{attribute 'qualified_only'}
VAR_GLOBAL
	Device_type															: ST_CAN_Object := (Name:='Device type', 														Index:=16#1000, 			 			Writeable:=FALSE);
	Error_register														: ST_CAN_Object := (Name:='Error register', 													Index:=16#1001, 			 Length:=1, Writeable:=FALSE);
	Manufacturer_status_register										: ST_CAN_Object := (Name:='Manufacturer status register', 										Index:=16#1002, 			 			Writeable:=FALSE);
	Pre_defined_error_field_Number_of_errors							: ST_CAN_Object := (Name:='Pre-defined error field_Number of errors',							Index:=16#1003, 			 Length:=1, 										SubElements:=E_SubElement_types.With_list);
	Pre_defined_error_field_Standard_error_field_1						: ST_CAN_Object := (Name:='Pre-defined error field_Standard error field 1',						Index:=16#1003, Subindex:=1, 			Writeable:=FALSE,						SubElements:=E_SubElement_types.List_element);
	COB_ID_SYNC															: ST_CAN_Object := (Name:='COB-ID SYNC',														Index:=16#1005, 			 			Writeable:=FALSE, Default_Value:=16#80);
	Communication_cycle_period											: ST_CAN_Object := (Name:='Communication cycle period',											Index:=16#1006);
	Synchronous_window_length											: ST_CAN_Object := (Name:='Synchronous window length',											Index:=16#1007);
	Manufacturer_device_name											: ST_CAN_Object := (Name:='Manufacturer device name', 											Index:=16#1008, 			 Length:=0, Writeable:=FALSE);
	Manufacturer_hardware_version										: ST_CAN_Object := (Name:='Manufacturer hardware version',										Index:=16#1009, 			 Length:=0, Writeable:=FALSE);
	Manufacturer_software_version										: ST_CAN_Object := (Name:='Manufacturer software version',										Index:=16#100A, 			 Length:=0, Writeable:=FALSE);
	Guard_time															: ST_CAN_Object := (Name:='Guard time', 														Index:=16#100C, 			 Length:=2, Writeable:=FALSE);
	Life_time_factor													: ST_CAN_Object := (Name:='Life time factor', 													Index:=16#100D, 			 Length:=1, Writeable:=FALSE);
	store_parameters_highest_sub_index_supported						: ST_CAN_Object := (Name:='store parameters_highest sub-index supported', 						Index:=16#1010, 			 Length:=1, Writeable:=FALSE, Default_Value:=4, 	SubElements:=E_SubElement_types.With_fix_subelements);
	store_parameters_save_all_parameters								: ST_CAN_Object := (Name:='store parameters_save all parameters', 								Index:=16#1010, Subindex:=1, 													SubElements:=E_SubElement_types.Fix_subelement);
	store_parameters_save_communication_parameters						: ST_CAN_Object := (Name:='store parameters_save communication parameters', 					Index:=16#1010, Subindex:=2, 													SubElements:=E_SubElement_types.Fix_subelement);
	store_parameters_save_application_parameters						: ST_CAN_Object := (Name:='store parameters_save application parameters', 						Index:=16#1010, Subindex:=3, 													SubElements:=E_SubElement_types.Fix_subelement);
	store_parameters_save_manufacture_label								: ST_CAN_Object := (Name:='store parameters_save manufacture label', 							Index:=16#1010, Subindex:=4, 													SubElements:=E_SubElement_types.Fix_subelement);
	restore_default_parameters_highest_sub_index_supported				: ST_CAN_Object := (Name:='restore default parameters_highest sub-index supported', 			Index:=16#1011, 			 Length:=1, Writeable:=FALSE, Default_Value:=4, 	SubElements:=E_SubElement_types.With_fix_subelements);
	restore_default_parameters_restore_all_default_parameters			: ST_CAN_Object := (Name:='restore default parameters_restore all default parameters', 			Index:=16#1011, Subindex:=1,													SubElements:=E_SubElement_types.Fix_subelement);
	restore_default_parameters_restore_communication_default_parameters	: ST_CAN_Object := (Name:='restore default parameters_restore communication default parameters',Index:=16#1011, Subindex:=2,													SubElements:=E_SubElement_types.Fix_subelement);
	restore_default_parameters_restore_application_default_parameters	: ST_CAN_Object := (Name:='restore default parameters_restore application default parameters', 	Index:=16#1011, Subindex:=3,													SubElements:=E_SubElement_types.Fix_subelement);
	restore_default_parameters_restore_default_manufacture_label		: ST_CAN_Object := (Name:='restore default parameters_restore default manufacture label', 		Index:=16#1011, Subindex:=4,													SubElements:=E_SubElement_types.Fix_subelement);
	COB_ID_time_stamp_message											: ST_CAN_Object := (Name:='COB-ID time stamp message', 											Index:=16#1012);
	High_resolution_time_stamp											: ST_CAN_Object := (Name:='High resolution time stamp', 										Index:=16#1013);
	COB_ID_emergency_message											: ST_CAN_Object := (Name:='COB-ID emergency message', 											Index:=16#1014);
	Inhibit_time_emergency_message										: ST_CAN_Object := (Name:='Inhibit time emergency message', 									Index:=16#1015, 			 Length:=2);
	Consumer_heartbeat_time_highest_sub_index_supported					: ST_CAN_Object := (Name:='Consumer heartbeat time_highest sub-index supported', 				Index:=16#1016, 			 Length:=1, 										SubElements:=E_SubElement_types.With_list);
	Consumer_heartbeat_time_1											: ST_CAN_Object := (Name:='Consumer heartbeat time 1',											Index:=16#1016, Subindex:=1, 													SubElements:=E_SubElement_types.List_element);
	Producer_heartbeat_time												: ST_CAN_Object := (Name:='Producer heartbeat time', 											Index:=16#1017, 			 Length:=2);
	Identity_object_Highest_sub_index_supported							: ST_CAN_Object := (Name:='Identity object_Highest sub-index supported', 						Index:=16#1018, 			 Length:=1, Writeable:=FALSE, Default_Value:=4, 	SubElements:=E_SubElement_types.With_fix_subelements);
	Identity_object_Vendor_ID											: ST_CAN_Object := (Name:='Identity object_Vendor-ID', 											Index:=16#1018, Subindex:=1, 			Writeable:=FALSE, 					 	SubElements:=E_SubElement_types.Fix_subelement);
	Identity_object_Product_code										: ST_CAN_Object := (Name:='Identity object_Product code',										Index:=16#1018, Subindex:=2, 			Writeable:=FALSE, 					 	SubElements:=E_SubElement_types.Fix_subelement);
	Identity_object_Revision_number										: ST_CAN_Object := (Name:='Identity object_Revision number',									Index:=16#1018, Subindex:=3, 			Writeable:=FALSE, 					 	SubElements:=E_SubElement_types.Fix_subelement);
	Identity_object_Serial_number										: ST_CAN_Object := (Name:='Identity object_Serial number',										Index:=16#1018, Subindex:=4, 			Writeable:=FALSE, 					 	SubElements:=E_SubElement_types.Fix_subelement);	
	Synchronous_counter_overflow_value									: ST_CAN_Object := (Name:='Synchronous counter overflow value', 								Index:=16#1019, 			 Length:=1);
	Verify_configuration_highest_sub_index_supported					: ST_CAN_Object := (Name:='Verify configuration_Highest sub-index supported', 					Index:=16#1020, 			 Length:=1, Writeable:=FALSE, Default_Value:=2, 	SubElements:=E_SubElement_types.With_fix_subelements);
	Verify_configuration_Configuration_date								: ST_CAN_Object := (Name:='Verify configuration_Configuration date', 							Index:=16#1020, Subindex:=1, 													SubElements:=E_SubElement_types.Fix_subelement);
	Verify_configuration_Configuration_time								: ST_CAN_Object := (Name:='Verify configuration_Configuration time', 							Index:=16#1020, Subindex:=2, 													SubElements:=E_SubElement_types.Fix_subelement);

	// SDO setting
	Server_SDO_Parameter_0_Number_of_entries							: ST_CAN_Object := (Name:='Server SDO Parameter 0_Number of entries', 							Index:=16#1200, 			 Length:=1, Writeable:=FALSE, Default_Value:=2, 	SubElements:=E_SubElement_types.With_fix_subelements);
	Server_SDO_Parameter_0_COB_ID_Client_to_Server						: ST_CAN_Object := (Name:='Server SDO Parameter 0_COB ID Client to Server', 					Index:=16#1200, Subindex:=1, 			Writeable:=FALSE,						SubElements:=E_SubElement_types.Fix_subelement);
	Server_SDO_Parameter_0_COB_ID_Server_to_Client						: ST_CAN_Object := (Name:='Server SDO Parameter 0_COB ID Server to Client', 					Index:=16#1200, Subindex:=2, 			Writeable:=FALSE,						SubElements:=E_SubElement_types.Fix_subelement);
	
	// PDO setting
	RPDO1_communication_parameter_Highest_sub_index_supported			: ST_CAN_Object := (Name:='RPDO communication parameter_Highest sub-index supported', 			Index:=16#1400, 			 Length:=1, Writeable:=FALSE, Default_Value:=5,		SubElements:=E_SubElement_types.With_fix_subelements);
	RPDO1_communication_parameter_COB_ID_used_by_RPDO					: ST_CAN_Object := (Name:='RPDO communication parameter_COB-ID used by RPDO', 					Index:=16#1400, Subindex:=1,													SubElements:=E_SubElement_types.Fix_subelement);
	RPDO1_communication_parameter_Transmission_type						: ST_CAN_Object := (Name:='RPDO communication parameter_Transmission type', 					Index:=16#1400, Subindex:=2, Length:=1, 										SubElements:=E_SubElement_types.Fix_subelement);
	RPDO1_communication_parameter_Event_timer							: ST_CAN_Object := (Name:='RPDO communication parameter_Event timer', 							Index:=16#1400, Subindex:=5, Length:=2, 										SubElements:=E_SubElement_types.Fix_subelement);
	RPDO2_communication_parameter_Highest_sub_index_supported			: ST_CAN_Object := (Name:='RPDO communication parameter_Highest sub-index supported',			Index:=16#1401, 			 Length:=1, Writeable:=FALSE, Default_Value:=5, 	SubElements:=E_SubElement_types.With_fix_subelements);
	RPDO2_communication_parameter_COB_ID_used_by_RPDO					: ST_CAN_Object := (Name:='RPDO communication parameter_COB-ID used by RPDO', 					Index:=16#1401, Subindex:=1,													SubElements:=E_SubElement_types.Fix_subelement);
	RPDO2_communication_parameter_Transmission_type						: ST_CAN_Object := (Name:='RPDO communication parameter_Transmission type', 					Index:=16#1401, Subindex:=2, Length:=1, 										SubElements:=E_SubElement_types.Fix_subelement);
	RPDO2_communication_parameter_Event_timer							: ST_CAN_Object := (Name:='RPDO communication parameter_Event timer', 							Index:=16#1401, Subindex:=5, Length:=2,											SubElements:=E_SubElement_types.Fix_subelement);
	RPDO3_communication_parameter_Highest_sub_index_supported			: ST_CAN_Object := (Name:='RPDO communication parameter_Highest sub-index supported', 			Index:=16#1402, 			 Length:=1, Writeable:=FALSE, Default_Value:=5, 	SubElements:=E_SubElement_types.With_fix_subelements);
	RPDO3_communication_parameter_COB_ID_used_by_RPDO					: ST_CAN_Object := (Name:='RPDO communication parameter_COB-ID used by RPDO', 					Index:=16#1402, Subindex:=1,													SubElements:=E_SubElement_types.Fix_subelement);
	RPDO3_communication_parameter_Transmission_type						: ST_CAN_Object := (Name:='RPDO communication parameter_Transmission type', 					Index:=16#1402, Subindex:=2, Length:=1, 										SubElements:=E_SubElement_types.Fix_subelement);
	RPDO3_communication_parameter_Event_timer							: ST_CAN_Object := (Name:='RPDO communication parameter_Event timer', 							Index:=16#1402, Subindex:=5, Length:=2,											SubElements:=E_SubElement_types.Fix_subelement);
	RPDO4_communication_parameter_Highest_sub_index_supported			: ST_CAN_Object := (Name:='RPDO communication parameter_Highest sub-index supported', 			Index:=16#1403, 			 Length:=1, Writeable:=FALSE, Default_Value:=5, 	SubElements:=E_SubElement_types.With_fix_subelements);
	RPDO4_communication_parameter_COB_ID_used_by_RPDO					: ST_CAN_Object := (Name:='RPDO communication parameter_COB-ID used by RPDO', 					Index:=16#1403, Subindex:=1,													SubElements:=E_SubElement_types.Fix_subelement);
	RPDO4_communication_parameter_Transmission_type						: ST_CAN_Object := (Name:='RPDO communication parameter_Transmission type', 					Index:=16#1403, Subindex:=2, Length:=1, 										SubElements:=E_SubElement_types.Fix_subelement);
	RPDO4_communication_parameter_Event_timer							: ST_CAN_Object := (Name:='RPDO communication parameter_Event timer', 							Index:=16#1403, Subindex:=5, Length:=2,											SubElements:=E_SubElement_types.Fix_subelement);
	RPDO1_mapping_parameter_Number_of_mapped_application_objects_in_PDO	: ST_CAN_Object := (Name:='RPDO mapping parameter_Number of mapped application objects in PDO', Index:=16#1600, 			 Length:=1, 										SubElements:=E_SubElement_types.With_fix_subelements);
	RPDO1_mapping_parameter_Application_object_1						: ST_CAN_Object := (Name:='RPDO mapping parameter_Application object 1', 						Index:=16#1600, Subindex:=1, 													SubElements:=E_SubElement_types.Fix_subelement);
	RPDO1_mapping_parameter_Application_object_2						: ST_CAN_Object := (Name:='RPDO mapping parameter_Application object 2', 						Index:=16#1600, Subindex:=2, 													SubElements:=E_SubElement_types.Fix_subelement);
	RPDO1_mapping_parameter_Application_object_3						: ST_CAN_Object := (Name:='RPDO mapping parameter_Application object 3', 						Index:=16#1600, Subindex:=3, 													SubElements:=E_SubElement_types.Fix_subelement);
	RPDO1_mapping_parameter_Application_object_4						: ST_CAN_Object := (Name:='RPDO mapping parameter_Application object 4', 						Index:=16#1600, Subindex:=4, 													SubElements:=E_SubElement_types.Fix_subelement);
	RPDO1_mapping_parameter_Application_object_5						: ST_CAN_Object := (Name:='RPDO mapping parameter_Application object 5', 						Index:=16#1600, Subindex:=5, 													SubElements:=E_SubElement_types.Fix_subelement);
	RPDO1_mapping_parameter_Application_object_6						: ST_CAN_Object := (Name:='RPDO mapping parameter_Application object 6',						Index:=16#1600, Subindex:=6, 													SubElements:=E_SubElement_types.Fix_subelement);
	RPDO1_mapping_parameter_Application_object_7						: ST_CAN_Object := (Name:='RPDO mapping parameter_Application object 7',						Index:=16#1600, Subindex:=7, 													SubElements:=E_SubElement_types.Fix_subelement);
	RPDO1_mapping_parameter_Application_object_8						: ST_CAN_Object := (Name:='RPDO mapping parameter_Application object 8', 						Index:=16#1600, Subindex:=8, 													SubElements:=E_SubElement_types.Fix_subelement);
	RPDO2_mapping_parameter_Number_of_mapped_application_objects_in_PDO	: ST_CAN_Object := (Name:='RPDO mapping parameter_Number of mapped application objects in PDO', Index:=16#1601, 			 Length:=1, 										SubElements:=E_SubElement_types.With_fix_subelements);
	RPDO2_mapping_parameter_Application_object_1						: ST_CAN_Object := (Name:='RPDO mapping parameter_Application object 1', 						Index:=16#1601, Subindex:=1, 													SubElements:=E_SubElement_types.Fix_subelement);
	RPDO2_mapping_parameter_Application_object_2						: ST_CAN_Object := (Name:='RPDO mapping parameter_Application object 2', 						Index:=16#1601, Subindex:=2, 													SubElements:=E_SubElement_types.Fix_subelement);
	RPDO2_mapping_parameter_Application_object_3						: ST_CAN_Object := (Name:='RPDO mapping parameter_Application object 3', 						Index:=16#1601, Subindex:=3, 													SubElements:=E_SubElement_types.Fix_subelement);
	RPDO2_mapping_parameter_Application_object_4						: ST_CAN_Object := (Name:='RPDO mapping parameter_Application object 4', 						Index:=16#1601, Subindex:=4, 													SubElements:=E_SubElement_types.Fix_subelement);
	RPDO2_mapping_parameter_Application_object_5						: ST_CAN_Object := (Name:='RPDO mapping parameter_Application object 5', 						Index:=16#1601, Subindex:=5, 													SubElements:=E_SubElement_types.Fix_subelement);
	RPDO2_mapping_parameter_Application_object_6						: ST_CAN_Object := (Name:='RPDO mapping parameter_Application object 6', 						Index:=16#1601, Subindex:=6, 													SubElements:=E_SubElement_types.Fix_subelement);
	RPDO2_mapping_parameter_Application_object_7						: ST_CAN_Object := (Name:='RPDO mapping parameter_Application object 7', 						Index:=16#1601, Subindex:=7, 													SubElements:=E_SubElement_types.Fix_subelement);
	RPDO2_mapping_parameter_Application_object_8						: ST_CAN_Object := (Name:='RPDO mapping parameter_Application object 8', 						Index:=16#1601, Subindex:=8, 													SubElements:=E_SubElement_types.Fix_subelement);
	RPDO3_mapping_parameter_Number_of_mapped_application_objects_in_PDO	: ST_CAN_Object := (Name:='RPDO mapping parameter_Number of mapped application objects in PDO', Index:=16#1602, 			 Length:=1, 										SubElements:=E_SubElement_types.With_fix_subelements);
	RPDO3_mapping_parameter_Application_object_1						: ST_CAN_Object := (Name:='RPDO mapping parameter_Application object 1', 						Index:=16#1602, Subindex:=1, 													SubElements:=E_SubElement_types.Fix_subelement);
	RPDO3_mapping_parameter_Application_object_2						: ST_CAN_Object := (Name:='RPDO mapping parameter_Application object 2', 						Index:=16#1602, Subindex:=2, 													SubElements:=E_SubElement_types.Fix_subelement);
	RPDO3_mapping_parameter_Application_object_3						: ST_CAN_Object := (Name:='RPDO mapping parameter_Application object 3', 						Index:=16#1602, Subindex:=3, 													SubElements:=E_SubElement_types.Fix_subelement);
	RPDO3_mapping_parameter_Application_object_4						: ST_CAN_Object := (Name:='RPDO mapping parameter_Application object 4', 						Index:=16#1602, Subindex:=4, 													SubElements:=E_SubElement_types.Fix_subelement);
	RPDO3_mapping_parameter_Application_object_5						: ST_CAN_Object := (Name:='RPDO mapping parameter_Application object 5', 						Index:=16#1602, Subindex:=5, 													SubElements:=E_SubElement_types.Fix_subelement);
	RPDO3_mapping_parameter_Application_object_6						: ST_CAN_Object := (Name:='RPDO mapping parameter_Application object 6', 						Index:=16#1602, Subindex:=6, 													SubElements:=E_SubElement_types.Fix_subelement);
	RPDO3_mapping_parameter_Application_object_7						: ST_CAN_Object := (Name:='RPDO mapping parameter_Application object 7', 						Index:=16#1602, Subindex:=7, 													SubElements:=E_SubElement_types.Fix_subelement);
	RPDO3_mapping_parameter_Application_object_8						: ST_CAN_Object := (Name:='RPDO mapping parameter_Application object 8', 						Index:=16#1602, Subindex:=8, 													SubElements:=E_SubElement_types.Fix_subelement);
	RPDO4_mapping_parameter_Number_of_mapped_application_objects_in_PDO	: ST_CAN_Object := (Name:='RPDO mapping parameter_Number of mapped application objects in PDO', Index:=16#1603, 			 Length:=1, 										SubElements:=E_SubElement_types.With_fix_subelements);
	RPDO4_mapping_parameter_Application_object_1						: ST_CAN_Object := (Name:='RPDO mapping parameter_Application object 1', 						Index:=16#1603, Subindex:=1, 													SubElements:=E_SubElement_types.Fix_subelement);
	RPDO4_mapping_parameter_Application_object_2						: ST_CAN_Object := (Name:='RPDO mapping parameter_Application object 2', 						Index:=16#1603, Subindex:=2, 													SubElements:=E_SubElement_types.Fix_subelement);
	RPDO4_mapping_parameter_Application_object_3						: ST_CAN_Object := (Name:='RPDO mapping parameter_Application object 3', 						Index:=16#1603, Subindex:=3, 													SubElements:=E_SubElement_types.Fix_subelement);
	RPDO4_mapping_parameter_Application_object_4						: ST_CAN_Object := (Name:='RPDO mapping parameter_Application object 4', 						Index:=16#1603, Subindex:=4, 													SubElements:=E_SubElement_types.Fix_subelement);
	RPDO4_mapping_parameter_Application_object_5						: ST_CAN_Object := (Name:='RPDO mapping parameter_Application object 5', 						Index:=16#1603, Subindex:=5, 													SubElements:=E_SubElement_types.Fix_subelement);
	RPDO4_mapping_parameter_Application_object_6						: ST_CAN_Object := (Name:='RPDO mapping parameter_Application object 6', 						Index:=16#1603, Subindex:=6, 													SubElements:=E_SubElement_types.Fix_subelement);
	RPDO4_mapping_parameter_Application_object_7						: ST_CAN_Object := (Name:='RPDO mapping parameter_Application object 7', 						Index:=16#1603, Subindex:=7, 													SubElements:=E_SubElement_types.Fix_subelement);
	RPDO4_mapping_parameter_Application_object_8						: ST_CAN_Object := (Name:='RPDO mapping parameter_Application object 8', 						Index:=16#1603, Subindex:=8, 													SubElements:=E_SubElement_types.Fix_subelement);
	TPDO1_communication_parameter_Highest_sub_index_supported			: ST_CAN_Object := (Name:='TPDO communication parameter_Highest sub-index supported', 			Index:=16#1800, 			 Length:=1, Writeable:=FALSE, Default_Value:=6, 	SubElements:=E_SubElement_types.With_fix_subelements);
	TPDO1_communication_parameter_COB_ID_used_by_TPDO					: ST_CAN_Object := (Name:='TPDO communication parameter_COB-ID used by TPDO', 					Index:=16#1800, Subindex:=1, 													SubElements:=E_SubElement_types.Fix_subelement);
	TPDO1_communication_parameter_Transmission_type						: ST_CAN_Object := (Name:='TPDO communication parameter_Transmission type', 					Index:=16#1800, Subindex:=2, Length:=1, 										SubElements:=E_SubElement_types.Fix_subelement);
	TPDO1_communication_parameter_Inhibit_time							: ST_CAN_Object := (Name:='TPDO communication parameter_Inhibit time', 							Index:=16#1800, Subindex:=3, Length:=2, 										SubElements:=E_SubElement_types.Fix_subelement);
	TPDO1_communication_parameter_Event_timer							: ST_CAN_Object := (Name:='TPDO communication parameter_Event timer', 							Index:=16#1800, Subindex:=5, Length:=2, 										SubElements:=E_SubElement_types.Fix_subelement);
	TPDO1_communication_parameter_SYNC_start_value						: ST_CAN_Object := (Name:='TPDO communication parameter_SYNC start value', 						Index:=16#1800, Subindex:=6, Length:=1, 										SubElements:=E_SubElement_types.Fix_subelement);						Index:=16#1800, Subindex:=6, Length:=1);	
	TPDO2_communication_parameter_Highest_sub_index_supported			: ST_CAN_Object := (Name:='TPDO communication parameter_Highest sub-index supported', 			Index:=16#1801, 			 Length:=1, Writeable:=FALSE, Default_Value:=6, 	SubElements:=E_SubElement_types.With_fix_subelements);
	TPDO2_communication_parameter_COB_ID_used_by_TPDO					: ST_CAN_Object := (Name:='TPDO communication parameter_COB-ID used by TPDO', 					Index:=16#1801, Subindex:=1, 													SubElements:=E_SubElement_types.Fix_subelement);
	TPDO2_communication_parameter_Transmission_type						: ST_CAN_Object := (Name:='TPDO communication parameter_Transmission type', 					Index:=16#1801, Subindex:=2, Length:=1, 										SubElements:=E_SubElement_types.Fix_subelement);
	TPDO2_communication_parameter_Inhibit_time							: ST_CAN_Object := (Name:='TPDO communication parameter_Inhibit time', 							Index:=16#1801, Subindex:=3, Length:=2, 										SubElements:=E_SubElement_types.Fix_subelement);
	TPDO2_communication_parameter_Event_timer							: ST_CAN_Object := (Name:='TPDO communication parameter_Event timer', 							Index:=16#1801, Subindex:=5, Length:=2, 										SubElements:=E_SubElement_types.Fix_subelement);
	TPDO2_communication_parameter_SYNC_start_value						: ST_CAN_Object := (Name:='TPDO communication parameter_SYNC start value', 						Index:=16#1801, Subindex:=6, Length:=1, 										SubElements:=E_SubElement_types.Fix_subelement);
	TPDO3_communication_parameter_Highest_sub_index_supported			: ST_CAN_Object := (Name:='TPDO communication parameter_Highest sub-index supported', 			Index:=16#1802, 			 Length:=1, Writeable:=FALSE, Default_Value:=6, 	SubElements:=E_SubElement_types.With_fix_subelements);
	TPDO3_communication_parameter_COB_ID_used_by_TPDO					: ST_CAN_Object := (Name:='TPDO communication parameter_COB-ID used by TPDO', 					Index:=16#1802, Subindex:=1, 													SubElements:=E_SubElement_types.Fix_subelement);
	TPDO3_communication_parameter_Transmission_type						: ST_CAN_Object := (Name:='TPDO communication parameter_Transmission type', 					Index:=16#1802, Subindex:=2, Length:=1, 										SubElements:=E_SubElement_types.Fix_subelement);
	TPDO3_communication_parameter_Inhibit_time							: ST_CAN_Object := (Name:='TPDO communication parameter_Inhibit time', 							Index:=16#1802, Subindex:=3, Length:=2, 										SubElements:=E_SubElement_types.Fix_subelement);
	TPDO3_communication_parameter_Event_timer							: ST_CAN_Object := (Name:='TPDO communication parameter_Event timer', 							Index:=16#1802, Subindex:=5, Length:=2, 										SubElements:=E_SubElement_types.Fix_subelement);
	TPDO3_communication_parameter_SYNC_start_value						: ST_CAN_Object := (Name:='TPDO communication parameter_SYNC start value', 						Index:=16#1802, Subindex:=6, Length:=1, 										SubElements:=E_SubElement_types.Fix_subelement);
	TPDO4_communication_parameter_Highest_sub_index_supported			: ST_CAN_Object := (Name:='TPDO communication parameter_Highest sub-index supported', 			Index:=16#1803, 			 Length:=1, Writeable:=FALSE, Default_Value:=6, 	SubElements:=E_SubElement_types.With_fix_subelements);
	TPDO4_communication_parameter_COB_ID_used_by_TPDO					: ST_CAN_Object := (Name:='TPDO communication parameter_COB-ID used by TPDO', 					Index:=16#1803, Subindex:=1, 													SubElements:=E_SubElement_types.Fix_subelement);
	TPDO4_communication_parameter_Transmission_type						: ST_CAN_Object := (Name:='TPDO communication parameter_Transmission type', 					Index:=16#1803, Subindex:=2, Length:=1, 										SubElements:=E_SubElement_types.Fix_subelement);
	TPDO4_communication_parameter_Inhibit_time							: ST_CAN_Object := (Name:='TPDO communication parameter_Inhibit time', 							Index:=16#1803, Subindex:=3, Length:=2, 										SubElements:=E_SubElement_types.Fix_subelement);
	TPDO4_communication_parameter_Event_timer							: ST_CAN_Object := (Name:='TPDO communication parameter_Event timer', 							Index:=16#1803, Subindex:=5, Length:=2, 										SubElements:=E_SubElement_types.Fix_subelement);
	TPDO4_communication_parameter_SYNC_start_value						: ST_CAN_Object := (Name:='TPDO communication parameter_SYNC start value', 						Index:=16#1803, Subindex:=6, Length:=1, 										SubElements:=E_SubElement_types.Fix_subelement);
	TPDO1_mapping_parameter_Number_of_mapped_application_objects_in_PDO	: ST_CAN_Object := (Name:='TPDO mapping parameter_Number of mapped application objects in PDO', Index:=16#1A00, 			 Length:=1, 										SubElements:=E_SubElement_types.With_fix_subelements);
	TPDO1_mapping_parameter_Application_object_1						: ST_CAN_Object := (Name:='TPDO mapping parameter_Application object 1', 						Index:=16#1A00, Subindex:=1, 													SubElements:=E_SubElement_types.Fix_subelement);
	TPDO1_mapping_parameter_Application_object_2						: ST_CAN_Object := (Name:='TPDO mapping parameter_Application object 2', 						Index:=16#1A00, Subindex:=2, 													SubElements:=E_SubElement_types.Fix_subelement);
	TPDO1_mapping_parameter_Application_object_3						: ST_CAN_Object := (Name:='TPDO mapping parameter_Application object 3', 						Index:=16#1A00, Subindex:=3, 													SubElements:=E_SubElement_types.Fix_subelement);
	TPDO1_mapping_parameter_Application_object_4						: ST_CAN_Object := (Name:='TPDO mapping parameter_Application object 4', 						Index:=16#1A00, Subindex:=4, 													SubElements:=E_SubElement_types.Fix_subelement);
	TPDO1_mapping_parameter_Application_object_5						: ST_CAN_Object := (Name:='TPDO mapping parameter_Application object 5',				 		Index:=16#1A00, Subindex:=5, 													SubElements:=E_SubElement_types.Fix_subelement);
	TPDO1_mapping_parameter_Application_object_6						: ST_CAN_Object := (Name:='TPDO mapping parameter_Application object 6', 						Index:=16#1A00, Subindex:=6, 													SubElements:=E_SubElement_types.Fix_subelement);
	TPDO1_mapping_parameter_Application_object_7						: ST_CAN_Object := (Name:='TPDO mapping parameter_Application object 7', 						Index:=16#1A00, Subindex:=7, 													SubElements:=E_SubElement_types.Fix_subelement);
	TPDO1_mapping_parameter_Application_object_8						: ST_CAN_Object := (Name:='TPDO mapping parameter_Application object 8',						Index:=16#1A00, Subindex:=8, 													SubElements:=E_SubElement_types.Fix_subelement);
	TPDO2_mapping_parameter_Number_of_mapped_application_objects_in_PDO	: ST_CAN_Object := (Name:='TPDO mapping parameter_Number of mapped application objects in PDO', Index:=16#1A01, 			 Length:=1,											SubElements:=E_SubElement_types.With_fix_subelements);
	TPDO2_mapping_parameter_Application_object_1						: ST_CAN_Object := (Name:='TPDO mapping parameter_Application object 1', 						Index:=16#1A01, Subindex:=1, 													SubElements:=E_SubElement_types.Fix_subelement);
	TPDO2_mapping_parameter_Application_object_2						: ST_CAN_Object := (Name:='TPDO mapping parameter_Application object 2', 						Index:=16#1A01, Subindex:=2, 													SubElements:=E_SubElement_types.Fix_subelement);
	TPDO2_mapping_parameter_Application_object_3						: ST_CAN_Object := (Name:='TPDO mapping parameter_Application object 3', 						Index:=16#1A01, Subindex:=3, 													SubElements:=E_SubElement_types.Fix_subelement);
	TPDO2_mapping_parameter_Application_object_4						: ST_CAN_Object := (Name:='TPDO mapping parameter_Application object 4', 						Index:=16#1A01, Subindex:=4, 													SubElements:=E_SubElement_types.Fix_subelement);
	TPDO2_mapping_parameter_Application_object_5						: ST_CAN_Object := (Name:='TPDO mapping parameter_Application object 5', 						Index:=16#1A01, Subindex:=5, 													SubElements:=E_SubElement_types.Fix_subelement);
	TPDO2_mapping_parameter_Application_object_6						: ST_CAN_Object := (Name:='TPDO mapping parameter_Application object 6', 						Index:=16#1A01, Subindex:=6, 													SubElements:=E_SubElement_types.Fix_subelement);
	TPDO2_mapping_parameter_Application_object_7						: ST_CAN_Object := (Name:='TPDO mapping parameter_Application object 7', 						Index:=16#1A01, Subindex:=7, 													SubElements:=E_SubElement_types.Fix_subelement);
	TPDO2_mapping_parameter_Application_object_8						: ST_CAN_Object := (Name:='TPDO mapping parameter_Application object 8', 						Index:=16#1A01, Subindex:=8, 													SubElements:=E_SubElement_types.Fix_subelement);
	TPDO3_mapping_parameter_Number_of_mapped_application_objects_in_PDO	: ST_CAN_Object := (Name:='TPDO mapping parameter_Number of mapped application objects in PDO', Index:=16#1A02, 			 Length:=1, 										SubElements:=E_SubElement_types.With_fix_subelements);
	TPDO3_mapping_parameter_Application_object_1						: ST_CAN_Object := (Name:='TPDO mapping parameter_Application object 1', 						Index:=16#1A02, Subindex:=1, 													SubElements:=E_SubElement_types.Fix_subelement);
	TPDO3_mapping_parameter_Application_object_2						: ST_CAN_Object := (Name:='TPDO mapping parameter_Application object 2', 						Index:=16#1A02, Subindex:=2, 													SubElements:=E_SubElement_types.Fix_subelement);
	TPDO3_mapping_parameter_Application_object_3						: ST_CAN_Object := (Name:='TPDO mapping parameter_Application object 3', 						Index:=16#1A02, Subindex:=3, 													SubElements:=E_SubElement_types.Fix_subelement);
	TPDO3_mapping_parameter_Application_object_4						: ST_CAN_Object := (Name:='TPDO mapping parameter_Application object 4', 						Index:=16#1A02, Subindex:=4, 													SubElements:=E_SubElement_types.Fix_subelement);
	TPDO3_mapping_parameter_Application_object_5						: ST_CAN_Object := (Name:='TPDO mapping parameter_Application object 5', 						Index:=16#1A02, Subindex:=5, 													SubElements:=E_SubElement_types.Fix_subelement);
	TPDO3_mapping_parameter_Application_object_6						: ST_CAN_Object := (Name:='TPDO mapping parameter_Application object 6', 						Index:=16#1A02, Subindex:=6, 													SubElements:=E_SubElement_types.Fix_subelement);
	TPDO3_mapping_parameter_Application_object_7						: ST_CAN_Object := (Name:='TPDO mapping parameter_Application object 7', 						Index:=16#1A02, Subindex:=7, 													SubElements:=E_SubElement_types.Fix_subelement);
	TPDO3_mapping_parameter_Application_object_8						: ST_CAN_Object := (Name:='TPDO mapping parameter_Application object 8', 						Index:=16#1A02, Subindex:=8, 													SubElements:=E_SubElement_types.Fix_subelement);
	TPDO4_mapping_parameter_Number_of_mapped_application_objects_in_PDO	: ST_CAN_Object := (Name:='TPDO mapping parameter_Number of mapped application objects in PDO', Index:=16#1A03, 			 Length:=1, 										SubElements:=E_SubElement_types.With_fix_subelements);
	TPDO4_mapping_parameter_Application_object_1						: ST_CAN_Object := (Name:='TPDO mapping parameter_Application object 1', 						Index:=16#1A03, Subindex:=1, 													SubElements:=E_SubElement_types.Fix_subelement);
	TPDO4_mapping_parameter_Application_object_2						: ST_CAN_Object := (Name:='TPDO mapping parameter_Application object 2', 						Index:=16#1A03, Subindex:=2, 													SubElements:=E_SubElement_types.Fix_subelement);
	TPDO4_mapping_parameter_Application_object_3						: ST_CAN_Object := (Name:='TPDO mapping parameter_Application object 3', 						Index:=16#1A03, Subindex:=3, 													SubElements:=E_SubElement_types.Fix_subelement);
	TPDO4_mapping_parameter_Application_object_4						: ST_CAN_Object := (Name:='TPDO mapping parameter_Application object 4', 						Index:=16#1A03, Subindex:=4, 													SubElements:=E_SubElement_types.Fix_subelement);
	TPDO4_mapping_parameter_Application_object_5						: ST_CAN_Object := (Name:='TPDO mapping parameter_Application object 5', 						Index:=16#1A03, Subindex:=5, 													SubElements:=E_SubElement_types.Fix_subelement);
	TPDO4_mapping_parameter_Application_object_6						: ST_CAN_Object := (Name:='TPDO mapping parameter_Application object 6', 						Index:=16#1A03, Subindex:=6, 													SubElements:=E_SubElement_types.Fix_subelement);
	TPDO4_mapping_parameter_Application_object_7						: ST_CAN_Object := (Name:='TPDO mapping parameter_Application object 7', 						Index:=16#1A03, Subindex:=7, 													SubElements:=E_SubElement_types.Fix_subelement);
	TPDO4_mapping_parameter_Application_object_8						: ST_CAN_Object := (Name:='TPDO mapping parameter_Application object 8', 						Index:=16#1A03, Subindex:=8, 													SubElements:=E_SubElement_types.Fix_subelement);
END_VAR

(* stored: Version 1.1.0.1, ProductVersion 3.1.4024.11
   GVL DS301_Object_List: Id {2975d994-08f1-4035-8338-1459181e384b} *)
